FUNCTION_BLOCK VAV_POST (* Variable Air Valve Model post-calculations *)
  (* Standard: 61499-1; Classification: Simulation; ApplicationDomain: HVAC; Function: Flow Sensor *)
  (* Version 0.0, 2006-04-10, JHC, Holobloc Inc *)
  (* Compiler header: package fb.rt.hvac; *)
  (* Compiler Java Sun JDK 1.5.0 *)
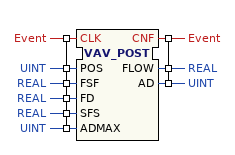
  EVENT_INPUT
    CLK WITH POS, FSF, SFS, FD, ADMAX; (* Perform post-model calculations *)
  END_EVENT
  EVENT_OUTPUT
    CNF WITH FLOW, AD; (* Post-calculations complete *)
  END_EVENT
  VAR_INPUT
    POS : UINT; (* Damper position, percent FS *)
    FSF : REAL := 1000.0; (* Air Flow at Damper Full Open, CFM *)
    FD : REAL; (* Maximum random flow deviation in CFM *)
    SFS : REAL := 1000.0; (* Air Flow at Sensor Full Scale, CFM *)
    ADMAX : UINT := 4096; (* Maximum Flow Sensor A/D converter value + 1, default is 12 bits *)
  END_VAR
  VAR_OUTPUT
    FLOW : REAL; (* Air flow, CFM *)
    AD : UINT; (* Flow sensor A/D converter value *)
  END_VAR
END_FUNCTION_BLOCK
